FUNCTION_BLOCK SUBSCRIBE_6
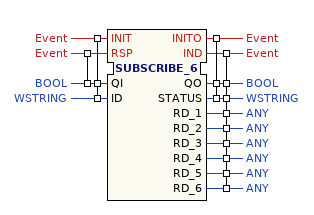
  EVENT_INPUT
    INIT WITH QI, ID;
    RSP WITH QI;
  END_EVENT
  EVENT_OUTPUT
    INITO WITH QO, STATUS;
    IND WITH QO, STATUS, RD_1, RD_3, RD_2, RD_4, RD_5, RD_6;
  END_EVENT
  VAR_INPUT
    QI : BOOL;
    ID : WSTRING;
  END_VAR
  VAR_OUTPUT
    QO : BOOL;
    STATUS : WSTRING;
    RD_1 : ANY;
    RD_2 : ANY;
    RD_3 : ANY;
    RD_4 : ANY;
    RD_5 : ANY;
    RD_6 : ANY;
  END_VAR
END_FUNCTION_BLOCK
